Staubli VAL3: setName.pgx

public program setName(string x_sName, num x_nIndex)
begin
  saveTool:name[x_nIndex]=x_sName
end
